FUNCTION TryConvert_DWORD_TO_UINT : BOOL
VAR_INPUT
	in : DWORD;
	out : REFERENCE TO UINT;
END_VAR

IF in > DatatypeLimits.MAX_VALUE_OF_DWORD_WHICH_CAN_BE_HELD_IN_A_UINT THEN
	RETURN;
END_IF

out := DWORD_TO_UINT(in);
TryConvert_DWORD_TO_UINT := TRUE;

END_FUNCTION

(* stored: Version 1.1.0.1, ProductVersion 3.1.4024.12
   POU TryConvert_DWORD_TO_UINT: Id {883f8311-3560-4d0e-909b-4eacf505cbe1}, SpecialFunc None *)
